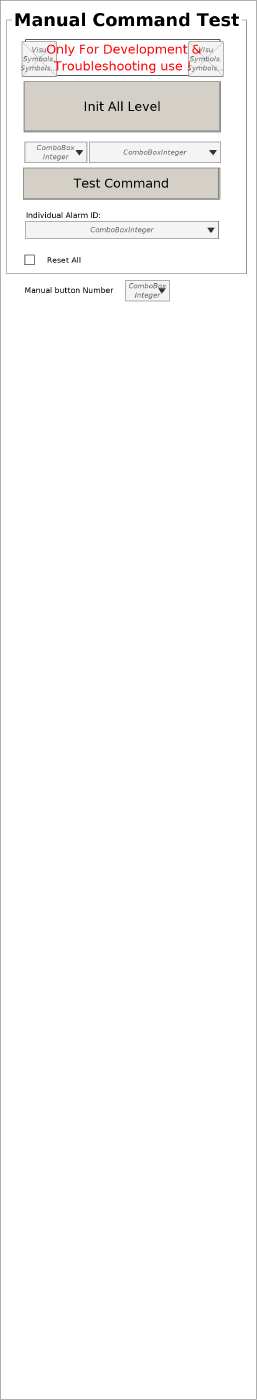
VISUALIZATION HMI_ManualCommand  // 367x1995
    Rectangle (9,-7 356x2000), invisible if: bEnableManualCommandTest1 AND bEnableManualCommandTest2
    GroupBox (9,20 343x370), "Manual Command Test"
        ComboBoxInteger (26,182 89x30), variable: iHMICbLevelSelection, text list: 'LevelTxtList'
    ComboBoxInteger (127,202 188x30), variable: iHMICbCmdSelection, text list: 'CmdTxtList'
    Button (33,239 281x45), "Test Command"
        tap TestManually.bTestCommand
    ComboBoxInteger (36,315 276x25), variable: TestManually.iAlarmCode, text list: 'AlarmTxtList'
    Checkbox (33,355 37x30), variable: bHMIResetAllAlarm
    Label (64,356 183x30), "Reset All"
    Label (34,292 215x30), "Individual Alarm ID:"
    Button (34,116 281x72), "Init All Level"
        tap TestManually.bInitialiseAll
    Rectangle (36,56 278x52)
    Image (31,59 50x50), image: VisuSymbols.Symbols.Caution
    Image (269,59 50x50), image: VisuSymbols.Symbols.Caution
    Label (63,56 221x29), "Only For Development &"
    Label (74,80 210x29), "Troubleshooting use !"
    ComboBoxInteger (179,399 63x30), variable: TestManually.iBtnNo
    Label (24,399 149x30), "Manual button Number"
END_VISUALIZATION

(* stored: Version 1.1.0.1, ProductVersion 3.1.4022.12
   Visu HMI_ManualCommand: Id {a78ecd60-a286-46be-a549-b88a79b8e299} *)
